FUNCTION_BLOCK AR_TO_AD_NUM (* Composite FB for numerically converting AR (REAL) adapter to AD (DWORD) adapter (via UDINT, not a bit-reinterpretation) *)
  (* Standard: 61499-2; Description: Copyright (c) 2026 HR Agrartechnik GmbH This program and the accompanying materials are made available under the terms of the Eclipse Public License 2.0 which is available at https://www.eclipse.org/legal/epl-2.0/ SPDX-License-Identifier: EPL-2.0 *)
  (* Version 1.0, 2026-09-07, Franz Höpfinger, HR Agrartechnik GmbH *)
  PACKAGE adapter::conversion::unidirectional;
  (* Documentation:
  AR_TO_AD_NUM
   🇩🇪 Deutsch
   Numerisch korrekte Alternative zu AR_TO_AD. Wandelt einen REAL-Adapter (AR_IN) über einen internen UDINT-Zwischenschritt in einen DWORD-Adapter (AD_OUT) um — echte Wertumwandlung, keine Bit-Reinterpretation. Die spiegelbildliche Ergänzung zu AD_TO_AR_NUM für die umgekehrte Richtung.
   Warum nicht einfach AR_TO_AD?
   AR_TO_AD nutzt intern F_REAL_TO_DWORD, was im FORTE-Kern für Bit-String-Zieltypen (DWORD/WORD/BYTE/LWORD) eine reine IEEE754-Bit-Reinterpretation ist, keinen numerischen Cast. Ein Sollwert wie REAL#50.0 würde dadurch NICHT zu DWORD#50, sondern zum rohen IEEE754-Bitmuster von 50.0 — als Tastgrad an einen PWM-Ausgang wie logiBUS_QDA_PWM gesendet also ein bedeutungsloser, weit außerhalb des gültigen Bereichs liegender Wert.
   AR_TO_AD_NUM vermeidet diese Falle, indem es zweistufig über F_REAL_TO_UDINT (echter numerischer Cast) und anschließend F_UDINT_TO_DWORD (Bit-Reinterpretation UDINT→DWORD, hier gültig, da beide dieselbe 32-bit-Darstellung eines vorzeichenlosen Integers teilen) konvertiert — dieselbe Kette, die auch von Hand über AR_TO_AUDI + AUDI_TO_AD verdrahtet werden kann (z.B. in Uebung_247_AX/Uebung_248_AX, PWM-Tastgrad-Ausgabe), hier als ein einziger, drop-in-kompatibler Baustein.
   Wann welchen Baustein verwenden?
    - AR_TO_AD_NUM: Der REAL-Wert ist eine Zahl (z. B. Prozent-Sollwert, PWM-Tastgrad) und soll als derselbe Zahlenwert in DWORD vorliegen (z.B. für einen logiBUS_QDA_PWM-Ausgang).
   - AR_TO_AD: Der REAL-Wert soll als IEEE754-Bitmuster serialisiert werden (z. B. zur Weitergabe an AD_TO_AR auf der Empfängerseite).
    🇬🇧 English
   Numerically correct alternative to AR_TO_AD. Converts a REAL adapter (AR_IN) into a DWORD adapter (AD_OUT) via an internal UDINT step — a real value conversion, not a bit-reinterpretation. The mirror-image counterpart to AD_TO_AR_NUM for the opposite direction.
   Why not just use AR_TO_AD?
   AR_TO_AD internally uses F_REAL_TO_DWORD, which in the FORTE core is a pure IEEE754 bit-reinterpretation for bit-string destination types (DWORD/WORD/BYTE/LWORD), not a numeric cast. A setpoint such as REAL#50.0 would NOT become DWORD#50 but the raw IEEE754 bit pattern of 50.0 — sent as a duty cycle to a PWM output such as logiBUS_QDA_PWM, a meaningless value far outside the valid range.
   AR_TO_AD_NUM avoids this trap by converting in two steps via F_REAL_TO_UDINT (a real numeric cast) and then F_UDINT_TO_DWORD (bit-reinterpretation UDINT→DWORD, valid here since both share the same 32-bit unsigned-integer representation) — the same chain that can also be wired by hand via AR_TO_AUDI + AUDI_TO_AD (e.g. in Uebung_247_AX/Uebung_248_AX, PWM duty-cycle output), packaged here as a single drop-in-compatible block.
   Which block to use?
    - AR_TO_AD_NUM: The REAL value is a number (e.g. a percent setpoint, PWM duty cycle) and should carry the same numeric value as DWORD (e.g. for a logiBUS_QDA_PWM output).
   - AR_TO_AD: The REAL value should be serialized as an IEEE754 bit pattern (e.g. to hand to AD_TO_AR on the receiving side).
  *)
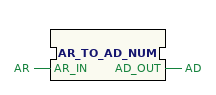
  SOCKETS
    AR_IN : adapter::types::unidirectional::AR; (* REAL Adapter Input *)
  END_SOCKETS
  PLUGS
    AD_OUT : adapter::types::unidirectional::AD; (* DWORD Adapter Output *)
  END_PLUGS
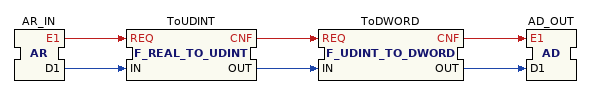
  FBS
    ToUDINT : iec61131::conversion::F_REAL_TO_UDINT;
    ToDWORD : iec61131::conversion::F_UDINT_TO_DWORD;
  END_FBS
  EVENT_CONNECTIONS
    AR_IN.E1 TO ToUDINT.REQ;
    ToUDINT.CNF TO ToDWORD.REQ;
    ToDWORD.CNF TO AD_OUT.E1;
  END_CONNECTIONS
  DATA_CONNECTIONS
    AR_IN.D1 TO ToUDINT.IN;
    ToUDINT.OUT TO ToDWORD.IN;
    ToDWORD.OUT TO AD_OUT.D1;
  END_CONNECTIONS
END_FUNCTION_BLOCK
